# EPICS IOC start-up script: test/startup/st.mcu010-SimCfg.iocsh
require ethercatmc,USER

epicsEnvSet("ECM_NUMAXES",   "6")
epicsEnvSet("MOTOR_PORT",    "$(SM_MOTOR_PORT=MCU1)")

epicsEnvSet("IPADDR",        "$(SM_IPADDR=127.0.0.1)")
epicsEnvSet("IPPORT",        "$(SM_IPPORT=5000)")
epicsEnvSet("ASYN_PORT",     "$(SM_ASYN_PORT=MC_CPU1)")
epicsEnvSet("PREFIX",        "$(SM_PREFIX=IOC:)")
epicsEnvSet("MOTOR_NAME",    "$(SM_MOTOR_NAME=m1)")
epicsEnvSet("AXIS_NO",       "$(SM_AXIS_NO=1)")
epicsEnvSet("DESC",          "$(SM_DESC=Lower=Right)")
epicsEnvSet("EGU",           "$(SM_EGU=mm)")
epicsEnvSet("PREC",          "$(SM_PREC=3)")

# And this reads the input of an incremental encoder terminal
# on the EtherCAT bus. Works with the simulator.
# For real terminals the adresses must be adapted
epicsEnvSet("AXISCONFIG",    "stepSize=1.0;HomProc=1;HomPos=-54;cfgFile=./mcu010-SoftSlit-1.cfg;encoder=ADSPORT=501/.ADR.16#3040010,16#80000049,2,2")

< ethercatmcController.iocsh
< ethercatmcAxis.iocsh
< ethercatmcAxisdebug.iocsh

epicsEnvSet("AXISCONFIG",    "stepSize=1.0;HomProc=2;HomPos=59;cfgFile=./mcu010-SoftSlit-2.cfg;encoder=ADSPORT=501/.ADR.16#3040010,16#8000004F,2,2")

epicsEnvSet("MOTOR_NAME",    "$(SM_MOTOR_NAME=m2)")
epicsEnvSet("AXIS_NO",       "$(SM_AXIS_NO=2)")
epicsEnvSet("DESC",          "$(SM_DESC=Upper=Left)")
< ethercatmcAxis.iocsh
< ethercatmcAxisdebug.iocsh

## Logical axes and slit
epicsEnvSet("P",             "$(PREFIX)")
epicsEnvSet("SLIT",          "$(SM_SLIT=SltH-)")
epicsEnvSet("mXp",           "$(SM_mXp=m2)")
epicsEnvSet("mXn",           "$(SM_mXp=m1)")
